FUNCTION_BLOCK F_MUX_32 (* multiplexer *)
  (* Standard: 61131-3; Classification: standard selection function; Description: Copyright (c) 2013 TU Wien ACIN\n \nThis program and the accompanying materials are made\navailable under the terms of the Eclipse Public License 2.0\nwhich is available at https://www.eclipse.org/legal/epl-2.0/\n\nSPDX-License-Identifier: EPL-2.0 *)
  (* Version 3.0, 2025-04-14, Patrick Aigner, changed package *)
  (* Version 1.1, 2024-07-15, Franz Höpfinger, HR Agrartechnik GmbH, F_MUX_3 copy and added 1 IN *)
  (* Version 1.0, 2013-08-30, Monika Wenger, TU Wien ACIN *)
  PACKAGE iec61131::selection;
  {SET_ATTRIBUTE(eclipse4diac::core::GenericClassName, 'GEN_F_MUX')}
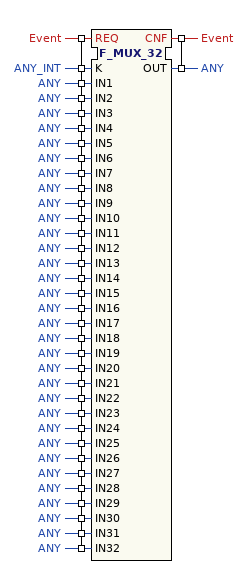
  EVENT_INPUT
    REQ WITH IN1, IN2, IN3, IN4, IN5, IN6, IN7, IN8, IN9, IN10, IN11, IN12, IN13, IN14, IN15, IN16, IN17, IN18, IN19, IN20, IN21, IN22, IN23, IN24, IN25, IN26, IN27, IN28, IN29, IN30, IN31, IN32, K; (* Service Request *)
  END_EVENT
  EVENT_OUTPUT
    CNF WITH OUT; (* Confirmation of Requested Service *)
  END_EVENT
  VAR_INPUT
    K : ANY_INT; (* Select one of n inputs *)
    IN1 : ANY; (* Input value 1 *)
    IN2 : ANY; (* Input value 2 *)
    IN3 : ANY; (* Input value 3 *)
    IN4 : ANY; (* Input value 4 *)
    IN5 : ANY; (* Input value 5 *)
    IN6 : ANY; (* Input value 6 *)
    IN7 : ANY; (* Input value 7 *)
    IN8 : ANY; (* Input value 8 *)
    IN9 : ANY; (* Input value 9 *)
    IN10 : ANY; (* Input value 10 *)
    IN11 : ANY; (* Input value 11 *)
    IN12 : ANY; (* Input value 12 *)
    IN13 : ANY; (* Input value 13 *)
    IN14 : ANY; (* Input value 14 *)
    IN15 : ANY; (* Input value 15 *)
    IN16 : ANY; (* Input value 16 *)
    IN17 : ANY; (* Input value 17 *)
    IN18 : ANY; (* Input value 18 *)
    IN19 : ANY; (* Input value 19 *)
    IN20 : ANY; (* Input value 20 *)
    IN21 : ANY; (* Input value 21 *)
    IN22 : ANY; (* Input value 22 *)
    IN23 : ANY; (* Input value 23 *)
    IN24 : ANY; (* Input value 24 *)
    IN25 : ANY; (* Input value 25 *)
    IN26 : ANY; (* Input value 26 *)
    IN27 : ANY; (* Input value 27 *)
    IN28 : ANY; (* Input value 28 *)
    IN29 : ANY; (* Input value 29 *)
    IN30 : ANY; (* Input value 30 *)
    IN31 : ANY; (* Input value 31 *)
    IN32 : ANY; (* Input value 32 *)
  END_VAR
  VAR_OUTPUT
    OUT : ANY; (* IN1 for K = 0, IN2 for K = 1, IN3 for K = 2, IN4 for K = 3, IN5 for K = 4, IN6 for K = 5, IN7 for K = 6, IN8 for K = 7, IN9 for K = 8, IN10 for K = 9, IN11 for K = 10, IN12 for K = 11, IN13 for K = 12, IN14 for K = 13, IN15 for K = 14, IN16 for K = 15, IN17 for K = 16, IN18 for K = 17, IN19 for K = 18, IN20 for K = 19, IN21 for K = 20, IN22 for K = 21, IN23 for K = 22, IN24 for K = 23, IN25 for K = 24, IN26 for K = 25, IN27 for K = 26, IN28 for K = 27, IN29 for K = 28, IN30 for K = 29, IN31 for K = 30, IN32 for K = 31 *)
  END_VAR
END_FUNCTION_BLOCK
